FUNCTION_BLOCK FB_ComponentEX EXTENDS FB_Component
VAR_INPUT
END_VAR
VAR_OUTPUT
END_VAR
VAR
	bEvent:			BOOL;
END_VAR

SUPER^();

METHOD PROTECTED M_Execute : BOOL
VAR_INPUT
END_VAR

IF bEvent THEN
	bEvent:= FALSE;
	fbEvent.M_Add('Test');
	fbEvent.M_Add('Test2');
	fbEvent.M_Add('Test3');
	fbEvent.M_Error('First Error Abort', 1 ,E_Behaviour.Abort);
END_IF
END_METHOD

END_FUNCTION_BLOCK

(* stored: Version 1.1.0.1, ProductVersion 3.1.4024.12
   POU FB_ComponentEX: Id {67ecce00-b6ba-4016-865f-4a4dfdc94a76}, SpecialFunc None
   Method M_Execute: Id {bba4d435-5736-45bd-97fd-4ceab6f0d012} *)
